{attribute 'GeneratedUsingTerminal: EK1100-0000-0018'}
{attribute addProperty BoxType "EK1100-0000-0018"}
{attribute addProperty Id "Beckhoff_EPP6xxxEK1122Beckhoff_EPP6xxxEK1122_AC5DD920594"}
{attribute addProperty CRC "3958060320"}
{attribute addProperty Size "594"}
TYPE Beckhoff_EPP6xxx_EBEB3520 EXTENDS EK1100_1FC0878B :
STRUCT
	{attribute addProperty Name "Beckhoff_EPP6xxxEK1122"}
	{attribute addProperty PreviousPort "Beckhoff EPP6xxx : B"}
	Beckhoff_EPP6xxxEK1122 : Beckhoff_EPP6xxxEK1122_AC5DD920;
END_STRUCT
END_TYPE

(* stored: Version 1.2.0.0, ProductVersion 3.1.4024.9
   DUT Beckhoff_EPP6xxx_EBEB3520: Id {4c479998-d452-4e11-b60e-5bc17b6d407e} *)
